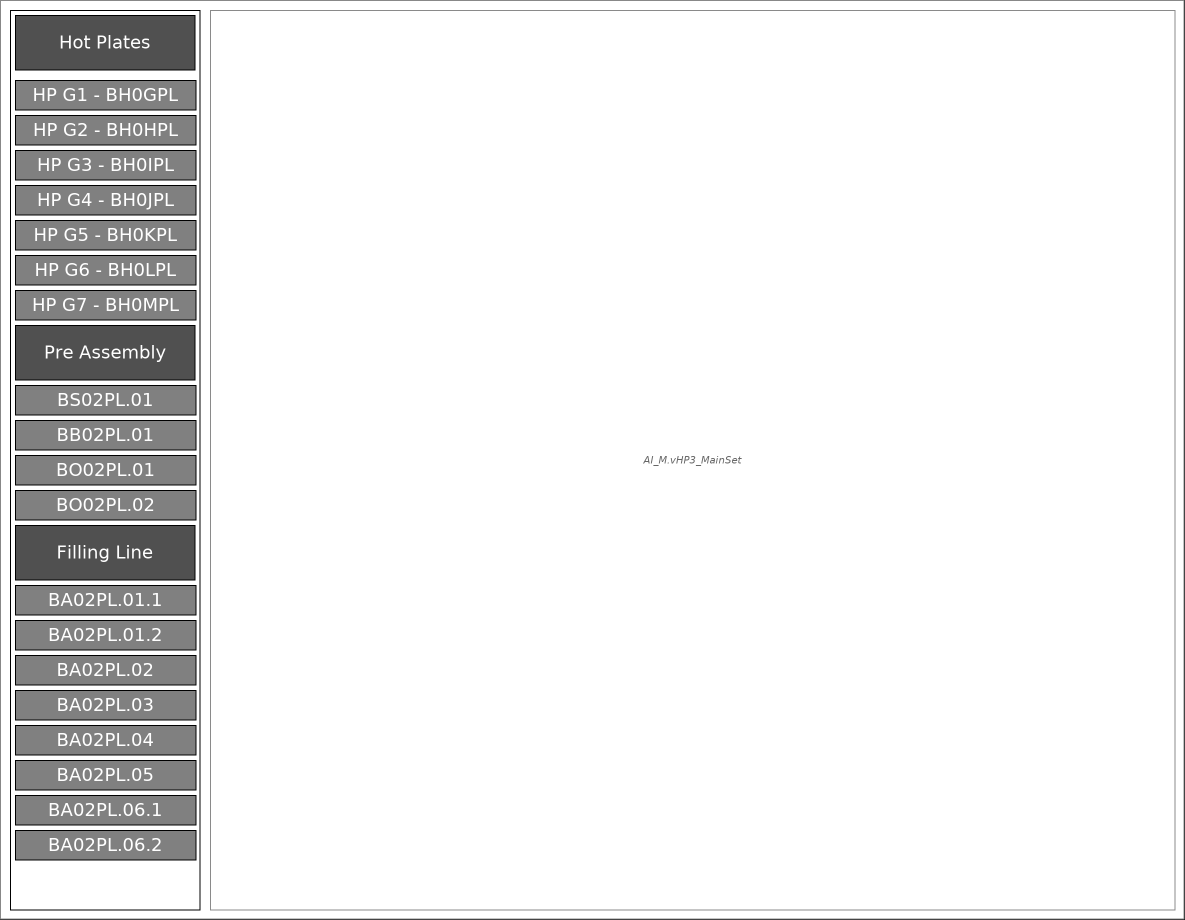
VISUALIZATION vHotPlateSettings_V3_B02PL  // 1185x920
VAR_IN_OUT
	fbHP1_M1	: fbHP_Control_V3_1;
	fbHP1_M2	: fbHP_Control_V3_1;
	fbHP1_M3	: fbHP_Control_V3_1;
	
	fbHP2_M1	: fbHP_Control_V3_1;
	fbHP2_M2	: fbHP_Control_V3_1;
	fbHP2_M3	: fbHP_Control_V3_1;
	
	fbHP3_M1	: fbHP_Control_V3_1;
	fbHP3_M2	: fbHP_Control_V3_1;
	fbHP3_M3	: fbHP_Control_V3_1;
	
	fbHP4_M1	: fbHP_Control_V3_1;
	fbHP4_M2	: fbHP_Control_V3_1;
	fbHP4_M3	: fbHP_Control_V3_1;
	
	fbHP5_M1	: fbHP_Control_V3_1;
	fbHP5_M2	: fbHP_Control_V3_1;
	fbHP5_M3	: fbHP_Control_V3_1;
	
	fbHP6_M1	: fbHP_Control_V3_1;
	fbHP6_M2	: fbHP_Control_V3_1;
	fbHP6_M3	: fbHP_Control_V3_1;
	
	fbHP7_M1	: fbHP_Control_V3_1;
	fbHP7_M2	: fbHP_Control_V3_1;
	fbHP7_M3	: fbHP_Control_V3_1;
	
	fbS01_Press						: fbSonicPress_V4_1;
	fbS01_FixtureBase				: fbSealingCorkAssKeyencePN_V4_1;
	
	fbS02_Press						: fbSonicPress_V4_1;
	
	fbS03_Press						: fbSonicPress_V4_1;
	fbS03_FixtureBase				: fbCapDetectionFixture_V4_1;
	
	fbS04_Press						: fbSonicPress_V4_1;
	
	stHMIData_Filler_A				:	stChiniseMachineHmiData_V3_1;
	stParams_Filler_A				:	stModTcpSlaveParams_V3_1;
	
	stHMIData_Cork					:	stChiniseMachineHmiData_V3_1;
	stParams_Cork					:	stModTcpSlaveParams_V3_1;
	
	stHMIData_Filler_B				:	stChiniseMachineHmiData_V3_1;
	stParams_Filler_B				:	stModTcpSlaveParams_V3_1;
	
	stHMIData_Sticker				:	stChiniseMachineHmiData_V3_1;
	stParams_Sticker				:	stModTcpSlaveParams_V3_1;
	
	stHMIData_Laser					:	stChiniseMachineHmiData_V3_2;
	stParams_Laser					:	stModTcpSlaveParams_V3_2;
	stHMI_Laser						: 	stHMI_Laser;
	
	fbSonic_S02						: fbSonictechUSWM_V4_1;
	
	fbSonic_S04						: fbSonictechUSWM_V4_1;
	
	fbVacuumChamber					: fbVacuumChamber_V3_2;
	fbTransporter					: fbTransporter_V3_2;
END_VAR
    Rectangle (0,0 1185x920)
    Frame (210,10 965x900)
        shows AI_M.vHP3_MainSet(fbHP_M1 := fbHP1_M1, fbHP_M2 := fbHP1_M2, fbHP_M3 := fbHP1_M3, NestNumber := 1, sSocketName := 'BH0GPL')
        shows AI_M.vHP3_MainSet(fbHP_M1 := fbHP2_M1, fbHP_M2 := fbHP2_M2, fbHP_M3 := fbHP2_M3, NestNumber := 2, sSocketName := 'BH0HPL')
        shows AI_M.vHP3_MainSet(fbHP_M1 := fbHP3_M1, fbHP_M2 := fbHP3_M2, fbHP_M3 := fbHP3_M3, NestNumber := 3, sSocketName := 'BH0IPL')
        shows AI_M.vHP3_MainSet(fbHP_M1 := fbHP4_M1, fbHP_M2 := fbHP4_M2, fbHP_M3 := fbHP4_M3, NestNumber := 4, sSocketName := 'BH0JPL')
        shows AI_M.vHP3_MainSet(fbHP_M1 := fbHP5_M1, fbHP_M2 := fbHP5_M2, fbHP_M3 := fbHP5_M3, NestNumber := 5, sSocketName := 'BH0KPL')
        shows AI_M.vHP3_MainSet(fbHP_M1 := fbHP6_M1, fbHP_M2 := fbHP6_M2, fbHP_M3 := fbHP6_M3, NestNumber := 6, sSocketName := 'BH0LPL')
        shows AI_M.vHP3_MainSet(fbHP_M1 := fbHP7_M1, fbHP_M2 := fbHP7_M2, fbHP_M3 := fbHP7_M3, NestNumber := 7, sSocketName := 'BH0MPL')
        shows AI_M.vSealingCorkAssPress_V4_1(fbData := fbS01_Press, fbFixtureBase := fbS01_FixtureBase)
        shows AI_M.vBaseSonicTechPress_V4_1(fbData := fbS02_Press)
        shows AI_M.vCapDetectionFixPress_V4_1(fbData := fbS03_Press, fbFixtureBase := fbS03_FixtureBase)
        shows AI_M.vBaseSonicTechPress_V4_1(fbData := fbS04_Press)
        shows AI_M.vChiniseMachineStatus_v3_1(stData := stHMIData_Filler_A, stParams := stParams_Filler_A)
        shows AI_M.vChiniseMachineStatus_v3_1(stData := stHMIData_Cork, stParams := stParams_Cork)
        shows AI_M.vBaseSonicTech_V4_1(fbData := fbSonic_S02)
        shows AI_M.vChiniseMachineStatus_v3_1(stData := stHMIData_Filler_B, stParams := stParams_Filler_B)
        shows AI_M.vBaseSonicTech_V4_1(fbData := fbSonic_S04)
        shows AI_M.vVacuumChamberMain_V3_2(fb := fbVacuumChamber, fbTrans := fbTransporter)
        shows AI_M.vChiniseMachineStatus_v3_1(stData := stHMIData_Sticker, stParams := stParams_Sticker)
        shows AI_M.vChiniseMachineStatus_Laser_V3_2(stData := stHMIData_Laser, stParams := stParams_Laser, stHMI_Laser := stHMI_Laser)
        shows vSetPacking_V3_Status_V3_2(fbData := fbS22)
        shows vDetectionTunelFrame_V3_1(stInOuts := stInOuts_Tunel, stParams := stParams_Tunel, iWorkStep := iWorkStep_Tunel, fb := fb_Tunel)
        p544952995: rS07HeaterTemperature
        p3767341414: fbS20
        p4018227088: fbS18.fbPIM
        p1625067722: fbS18.stHwSettings
        p4124004121: fbS18.stInOuts.iPressure
        p961079038: fbS16.stInOuts
        p1151590893: fbSonic_S16
        p2539462775: fbS14
        p3846459017: fbS11.fbPIM
        p39883683: fbS10
        p445293019: fbSonic_S10
        p2875566315: fbS10.stInOuts
        p426879848: fbSonic_S09.fbPIM.stStation.sStationName
        p268622539: fbS06.stSettings
        p836702480: fbS06.stInOuts
        p773328817: fbSonic_S06.stDigitalInOut
        p11944277: fbSonic_S06
        p847402520: fbS07.stInOuts.rHeatStampTemperature
    Rectangle (10,10 190x900)
    Rectangle (15,80 181x30), "HP G1 - BH0GPL"
        OnMouseDown: FrameSelectionChange Selection=SelectedFrame=2676ba61-b932-4ea5-9074-f1d3beec8c67, GlobSel=AssignType=Directly, SelType=Locally
    Rectangle (15,15 180x55), "Hot Plates"
    Rectangle (15,115 181x30), "HP G2 - BH0HPL"
        OnMouseDown: FrameSelectionChange Selection=SelectedFrame=2676ba61-b932-4ea5-9074-f1d3beec8c67, Selection=1, GlobSel=AssignType=Directly, SelType=Locally
    Rectangle (15,255 181x30), "HP G6 - BH0LPL"
        OnMouseDown: FrameSelectionChange Selection=SelectedFrame=2676ba61-b932-4ea5-9074-f1d3beec8c67, Selection=5, GlobSel=AssignType=Directly, SelType=Locally
    Rectangle (15,185 181x30), "HP G4 - BH0JPL"
        OnMouseDown: FrameSelectionChange Selection=SelectedFrame=2676ba61-b932-4ea5-9074-f1d3beec8c67, Selection=3, GlobSel=AssignType=Directly, SelType=Locally
    Rectangle (15,290 181x30), "HP G7 - BH0MPL"
        OnMouseDown: FrameSelectionChange Selection=SelectedFrame=2676ba61-b932-4ea5-9074-f1d3beec8c67, Selection=6, GlobSel=AssignType=Directly, SelType=Locally
    Rectangle (15,325 180x55), "Pre Assembly"
    Rectangle (15,385 181x30), "BS02PL.01"
        OnMouseDown: FrameSelectionChange Selection=SelectedFrame=2676ba61-b932-4ea5-9074-f1d3beec8c67, Selection=7, GlobSel=AssignType=Directly, SelType=Locally
    Rectangle (15,150 181x30), "HP G3 - BH0IPL"
        OnMouseDown: FrameSelectionChange Selection=SelectedFrame=2676ba61-b932-4ea5-9074-f1d3beec8c67, Selection=2, GlobSel=AssignType=Directly, SelType=Locally
    Rectangle (15,455 181x30), "BO02PL.01"
        OnMouseDown: FrameSelectionChange Selection=SelectedFrame=2676ba61-b932-4ea5-9074-f1d3beec8c67, Selection=9, GlobSel=AssignType=Directly, SelType=Locally
    Rectangle (15,420 181x30), "BB02PL.01"
        OnMouseDown: FrameSelectionChange Selection=SelectedFrame=2676ba61-b932-4ea5-9074-f1d3beec8c67, Selection=8, GlobSel=AssignType=Directly, SelType=Locally
    Rectangle (15,490 181x30), "BO02PL.02"
        OnMouseDown: FrameSelectionChange Selection=SelectedFrame=2676ba61-b932-4ea5-9074-f1d3beec8c67, Selection=10, GlobSel=AssignType=Directly, SelType=Locally
    Rectangle (15,690 181x30), "BA02PL.03"
        OnMouseDown: FrameSelectionChange Selection=SelectedFrame=2676ba61-b932-4ea5-9074-f1d3beec8c67, Selection=14, GlobSel=AssignType=Directly, SelType=Locally
    Rectangle (15,620 181x30), "BA02PL.01.2"
        OnMouseDown: FrameSelectionChange Selection=SelectedFrame=2676ba61-b932-4ea5-9074-f1d3beec8c67, Selection=12, GlobSel=AssignType=Directly, SelType=Locally
    Rectangle (15,585 181x30), "BA02PL.01.1"
        OnMouseDown: FrameSelectionChange Selection=SelectedFrame=2676ba61-b932-4ea5-9074-f1d3beec8c67, Selection=11, GlobSel=AssignType=Directly, SelType=Locally
    Rectangle (15,655 181x30), "BA02PL.02"
        OnMouseDown: FrameSelectionChange Selection=SelectedFrame=2676ba61-b932-4ea5-9074-f1d3beec8c67, Selection=13, GlobSel=AssignType=Directly, SelType=Locally
    Rectangle (15,220 181x30), "HP G5 - BH0KPL"
        OnMouseDown: FrameSelectionChange Selection=SelectedFrame=2676ba61-b932-4ea5-9074-f1d3beec8c67, Selection=4, GlobSel=AssignType=Directly, SelType=Locally
    Rectangle (15,525 180x55), "Filling Line"
    Rectangle (15,830 181x30), "BA02PL.06.2"
        OnMouseDown: FrameSelectionChange Selection=SelectedFrame=2676ba61-b932-4ea5-9074-f1d3beec8c67, Selection=18, GlobSel=AssignType=Directly, SelType=Locally
    Rectangle (15,760 181x30), "BA02PL.05"
        OnMouseDown: FrameSelectionChange Selection=SelectedFrame=2676ba61-b932-4ea5-9074-f1d3beec8c67, Selection=16, GlobSel=AssignType=Directly, SelType=Locally
    Rectangle (15,725 181x30), "BA02PL.04"
        OnMouseDown: FrameSelectionChange Selection=SelectedFrame=2676ba61-b932-4ea5-9074-f1d3beec8c67, Selection=15, GlobSel=AssignType=Directly, SelType=Locally
    Rectangle (15,795 181x30), "BA02PL.06.1"
        OnMouseDown: FrameSelectionChange Selection=SelectedFrame=2676ba61-b932-4ea5-9074-f1d3beec8c67, Selection=17, GlobSel=AssignType=Directly, SelType=Locally
END_VISUALIZATION

(* stored: Version 1.1.0.1, ProductVersion 3.1.4024.16
   Visu vHotPlateSettings_V3_B02PL: Id {c9dcf8e5-0ffc-452d-ace2-286d928724b6} *)
